// Mitsubishi GX Works2 project: LRI - PLC - AULA 11   PLC: Q03UDV

// task Task_01 (event TRUE, interval 0, priority 31): POU_01

PROGRAM POU_01
END_PROGRAM

PROGRAM ST_Exemplo
VAR
  iDR : ARRAY [0..3] OF INT;  (* Declaração de varivavel ST *)
END_VAR
VAR CONSTANT
  iElemento01 : INT := 15;
  iElemento02 : INT := 4;
END_VAR



iDR[0] :=iElemento01 + iElemento02;
iDR[1] :=iElemento01 - iElemento02;
iDR[2] :=iElemento01 * iElemento02;
iDR[3] :=iElemento01 MOD(iElemento01,iElemento02);
END_PROGRAM
